Staubli VAL3: next.pgx

public program next(string x_sItem)
  local num l_nValue
  local num l_nSize
begin
  // get the actual position
  call getPalletPos(x_sItem,l_nValue)
  call getSizePallet(x_sItem,l_nSize)
  // go to the next ONE
  if l_nValue<l_nSize-1
    call setPalletPos(x_sItem,l_nValue+1)
  else
    call setPalletPos(x_sItem,0)
  endIf
end
